FUNCTION init_Grn : BOOL
VAR_INPUT
	pGrn			: POINTER TO T_GRN;
	/// instance array of all controller instances
	pCtrlInst		: POINTER TO fb_CtrlBase;
	/// common interface array of all controllers (main use for PLC)
	pCtrlCIf		: POINTER TO T_Ctrl_CIf;
END_VAR

pGrn^.ctrl.fbGrn.iniAllCtrlArrays(pCtrlInst,pCtrlCIf,pGrn^.id.Grn);

END_FUNCTION

(* stored: Version 1.1.0.1, ProductVersion 3.1.0.25
   POU init_Grn: Id {28c11cc5-75dd-4c5f-9183-c6956d5e8d7a} *)
